// TIA Portal project "Elementary_data_types-ScopeDB" (V16)

(* hardware
DEVICE "S71500/ET200MP station_1"  S7-1500 station
   slot 0: "Rail_0"  Rack  6ES7 590-1***0-0AA0
   slot 1: "PLC_1"  CPU 1511F-1 PN  6ES7 511-1FK02-0AB0  V2.8
      slot 3: "CPU display_1"  6ES7591-1AA00-0AA0
      slot 32768: "PROFINET interface_1"  X1
      slot 34817: "Virtual CP interface port_1"  Virtual CP interface port  Virtual CP interface port
*)

// ===== PLC "PLC_1"  CPU 1511F-1 PN =====

// folder: Elementary data types

DATA_BLOCK "Binary numbers"   // DB1
{ S7_Optimized_Access := 'TRUE' }
VERSION : 0.1
   VAR
      DB_Bool : Bool;
      DB_Byte : Byte;
      DB_Word : Word;
      DB_Dword : DWord;
      DB_LWord : LWord;
   END_VAR
BEGIN
END_DATA_BLOCK

DATA_BLOCK "Integers"   // DB2
{ S7_Optimized_Access := 'TRUE' }
VERSION : 0.1
   VAR
      DB_Sint : SInt;
      DB_Int : Int;
      DB_Dint : DInt;
      DB_Usint : USInt;
      DB_Uint : UInt;
      DB_Udint : UDInt;
      DB_Lint : LInt;
      DB_Ulint : ULInt;
   END_VAR
BEGIN
END_DATA_BLOCK

DATA_BLOCK "Floating-point numbers"   // DB3
{ S7_Optimized_Access := 'TRUE' }
VERSION : 0.1
   VAR
      DB_Real : Real;
      DB_Lreal : LReal;
   END_VAR
BEGIN
END_DATA_BLOCK

DATA_BLOCK "Timers"   // DB4
{ S7_Optimized_Access := 'TRUE' }
VERSION : 0.1
   VAR
      DB_S5Time : S5Time;
      DB_Time : Time;
      DB_Ltime : LTime;
   END_VAR
BEGIN
END_DATA_BLOCK

DATA_BLOCK "Datetime_Char"   // DB5
{ S7_Optimized_Access := 'TRUE' }
VERSION : 0.1
   VAR
      DB_Date : Date;
      DB_Tod : Time_Of_Day;
      DB_Ltod : LTime_Of_Day;
      DB_Char : Char;
      DB_Wchar : WChar;
   END_VAR
BEGIN
END_DATA_BLOCK

DATA_BLOCK "Character strings"   // DB6
{ S7_Optimized_Access := 'TRUE' }
VERSION : 0.1
   VAR
      DB_Char : Char;
      DB_WChar : WChar;
   END_VAR
BEGIN
END_DATA_BLOCK

// folder: (top level)

ORGANIZATION_BLOCK "Main"   // OB1, LAD, ProgramCycle
TITLE = "Main Program Sweep (Cycle)"
{ S7_Optimized_Access := 'TRUE' }
VERSION : 0.1
   VAR_INPUT
      Initial_Call : Bool;   // Initial call of this OB
      Remanence : Bool;   // =True, if remanent data are available
   END_VAR
BEGIN
END_ORGANIZATION_BLOCK